(* IEC 61131-3 sources: F100R_S278_Temperville/MyController.device.xml.v3^/Plc Logic.plclogic.xml.v3^/Application.application.xml.v3^/06_Relógio, 3 files *)

(* ---- B_DataHora.prg.st ---- *)
PROGRAM B_DataHora
VAR
	LerDataHora: GetDateAndTime;
	SetDataHora: SetDateAndTime;
	TonAcertoHora: TON;
	TonAcertoHoraIn: BOOL;
	TonAcertoHoraQ: BOOL;
	uAnoRealTimeq_UIntMonth: UINT;
END_VAR

// Auto Acerto Data/Hora

TonAcertoHoraIn:= NOT TonAcertoHoraQ;

TonAcertoHora(IN:= TonAcertoHoraIn, PT:=T#30S , Q=>TonAcertoHoraQ, ET=> );

IF TonAcertoHoraQ THEN
	xAcertaRelogio:=TRUE;
END_IF

SetDataHora(
	i_xSetDateTime:= 	BtAcertaRelogioPlc,
	i_UIntYear:= 		uAcertoAno,
	i_UIntMonth:= 		uAcertoMes,
	i_UIntDay:= 		uAcertoDia,
	i_UIntHour:= 		uAcertoHora,
	i_UIntMinute:= 		uAcertoMinuto,
	i_UIntSecond:= 		uAcertoSegundo,
	q_UIntDatetoUTC_diag=> ,
	q_UIntRtcSet_diag=> );

IF BtAcertaRelogioPlc THEN
	BtAcertaRelogioPlc:=false;
END_IF

LerDataHora(
	q_UIntYear=> 		uAnoRealTime,
	q_UIntMonth=> 		uMesRealTime,
	q_UIntDay=> 		uDiaRealTime,
	q_UIntHour=> 		uHoraRealTime,
	q_UIntMinute=> 		uMinutoRealTime,
	q_UIntSecond=> 		uSegundoRealTime,
	q_UIntMSecond=> 	uMSegundoRealTime,
	q_UIntDayOfWeek=> 	uDiaSemanaRealTime,
	q_UIntYday=> 		uDiaAnoRealTime);

IF xRelogioAcertado THEN
	xAcertaRelogio:=FALSE;
	xRelogioAcertado:=FALSE;
END_IF

(* ---- C_ProgramacaoHoraria.prg.st ---- *)
PROGRAM C_ProgramacaoHoraria
VAR
	AtivaDesativaSemanal: HabilitaDesabilita;
	AtivaDesativaDiaria: HabilitaDesabilita;
	xLigaSegunda: BOOL;
	xLigaTerca: BOOL;
	xLigaQuarta: BOOL;
	xLigaQuinta: BOOL;
	xLigaSexta: BOOL;
	xLigaSabado: BOOL;
	xLigaDomingo: BOOL;
	xLigaSemanda: BOOL;

	xLigaHoraSeg: BOOL;
	xLigaMinutoSeg: BOOL;
	xLigaHoraTer: BOOL;
	xLigaMinutoTer: BOOL;
	xLigaHoraQua: BOOL;
	xLigaMinutoQua: BOOL;
	xLigaHoraQui: BOOL;
	xLigaMinutoQui: BOOL;
	xLigaHoraSex: BOOL;
	xLigaMinutoSex: BOOL;
	xLigaHoraSab: BOOL;
	xLigaMinutoSab: BOOL;
	xLigaHoraDom: BOOL;
	xLigaMinutoDom: BOOL;
	xLigaSegundo: BOOL;
	xLigaTempoSeg: BOOL;
	xLigaTempoTer: BOOL;
	xLigaTempoQua: BOOL;
	xLigaTempoQui: BOOL;
	xLigaTempoSex: BOOL;
	xLigaTempoSab: BOOL;
	xLigaTempoDom: BOOL;
	xLigaSemanaDias: BOOL;
	uDiaSemanaRealTimeAuxiliar: UINT;
	xAuxLiga: BOOL;
	xAuxEnable: BOOL;
	teste: BOOL;

	xDataHoraDomProgOk	: BOOL ;
	xDataHoraSegProgOk	: BOOL ;
	xDataHoraTerProgOk	: BOOL ;
	xDataHoraQuaProgOk	: BOOL ;
	xDataHoraQuiProgOk	: BOOL ;
	xDataHoraSexProgOk	: BOOL ;
	xDataHoraSabProgOk	: BOOL ;

END_VAR

// Programação Horario

IF uDiaSemanaRealTime=0 THEN
	uDiaSemanaRealTimeAuxiliar:=7;
ELSE
	uDiaSemanaRealTimeAuxiliar:=uDiaSemanaRealTime;
END_IF

//Horario Domingo
xLigaHoraDom:=		uHoraRealTime = rHorProgramadoDom;
xLigaMinutoDom:=	uMinutoRealTime = rMinProgramadoDom;
xLigaSegundo:=		uSegundoRealTime = uSegProgramado;
xLigaTempodom := xLigaHoraDom AND xLigaMinutoDom AND xLigaSegundo;

IF bDomingo AND uDiaSemanaRealTimeAuxiliar=7 THEN
	xLigaDomingo:=TRUE;
ELSE
	xLigaDomingo:=FALSE;
END_IF

xDataHoraDomProgOk:= xLigaDomingo AND xLigaTempodom;
IF xDataHoraDomProgOk THEN
	rTempoRampa03 := rRampaDomingo;
END_IF

//Horario Segunda
xLigaHoraSeg:=		uHoraRealTime = rHorProgramadoSeg;
xLigaMinutoSeg:=	uMinutoRealTime = rMinProgramadoSeg;
xLigaSegundo:=		uSegundoRealTime = uSegProgramado;
xLigaTempoSeg := xLigaHoraSeg AND xLigaMinutoSeg AND xLigaSegundo;

IF bSegunda AND uDiaSemanaRealTimeAuxiliar=1 THEN
	xLigaSegunda:=TRUE;
ELSE
	xLigaSegunda:=FALSE;
END_IF

xDataHoraSegProgOk:= xLigaSegunda AND xLigaTempoSeg;
IF xDataHoraSegProgOk THEN
	rTempoRampa03 := rRampaSegunda;
END_IF

//Horario Terça
xLigaHoraTer:=		uHoraRealTime = rHorProgramadoTer;
xLigaMinutoTer:=	uMinutoRealTime = rMinProgramadoTer;
xLigaSegundo:=		uSegundoRealTime = uSegProgramado;
xLigaTempoTer := xLigaHoraTer AND xLigaMinutoTer AND xLigaSegundo;

IF bTerca AND uDiaSemanaRealTimeAuxiliar=2 THEN
	xLigaTerca:=TRUE;
ELSE
	xLigaTerca:=FALSE;
END_IF

xDataHoraTerProgOk:= xLigaTerca AND xLigaTempoTer;
IF xDataHoraTerProgOk THEN
	rTempoRampa03 := rRampaTerca;
END_IF
//Horario Quarta
xLigaHoraQua:=		uHoraRealTime = rHorProgramadoQua;
xLigaMinutoQua:=	uMinutoRealTime = rMinProgramadoQua;
xLigaSegundo:=		uSegundoRealTime = uSegProgramado;
xLigaTempoQua := xLigaHoraQua AND xLigaMinutoQua AND xLigaSegundo;

IF bQuarta AND uDiaSemanaRealTimeAuxiliar=3 THEN
	xLigaQuarta:=TRUE;
ELSE
	xLigaQuarta:=FALSE;
END_IF

xDataHoraQuaProgOk:= xLigaQuarta AND xLigaTempoQua;
IF xDataHoraQuaProgOk THEN
	rTempoRampa03 := rRampaQuarta;
END_IF

//Horario Quinta
xLigaHoraQui:=		uHoraRealTime = rHorProgramadoQui;
xLigaMinutoQui:=	uMinutoRealTime = rMinProgramadoQui;
xLigaSegundo:=		uSegundoRealTime = uSegProgramado;
xLigaTempoQui := xLigaHoraQui AND xLigaMinutoQui AND xLigaSegundo;

IF bQuinta AND uDiaSemanaRealTimeAuxiliar=4 THEN
	xLigaQuinta:=TRUE;
ELSE
	xLigaQuinta:=FALSE;
END_IF

xDataHoraQuiProgOk:= xLigaQuinta AND xLigaTempoQui;
IF xDataHoraQuiProgOk THEN
	rTempoRampa03 := rRampaQuinta;
END_IF

//Horario Sexta
xLigaHoraSex:=		uHoraRealTime = rHorProgramadoSex;
xLigaMinutoSex:=	uMinutoRealTime = rMinProgramadoSex;
xLigaSegundo:=		uSegundoRealTime = uSegProgramado;
xLigaTempoSex := xLigaHoraSex AND xLigaMinutoSex AND xLigaSegundo;

IF bSexta AND uDiaSemanaRealTimeAuxiliar=5 THEN
	xLigaSexta:=TRUE;
ELSE
	xLigaSexta:=FALSE;
END_IF

xDataHoraSexProgOk:= xLigaSexta AND xLigaTempoSex;
IF xDataHoraSexProgOk THEN
	rTempoRampa03 := rRampaSexta;
END_IF

//Horario Sabado
xLigaHoraSab:=		uHoraRealTime = rHorProgramadoSab;
xLigaMinutoSab:=	uMinutoRealTime = rMinProgramadoSab;
xLigaSegundo:=		uSegundoRealTime = uSegProgramado;
xLigaTempoSab := 	xLigaHoraSab AND xLigaMinutoSab AND xLigaSegundo;

IF bSabado AND uDiaSemanaRealTimeAuxiliar=6 THEN
	xLigaSabado:=TRUE;
ELSE
	xLigaSabado:=FALSE;
END_IF

xDataHoraSabProgOk:= xLigaSabado AND xLigaTempoSab;
IF xDataHoraSabProgOk THEN
	rTempoRampa03 := rRampaSabado;
END_IF

// Programação Horaria Ativada

IF bDomingo OR bSegunda OR bTerca OR bQuarta OR bQuinta OR bSexta OR bSabado THEN
	bStatusAtvProgSemana:=TRUE;
ELSE
	bStatusAtvProgSemana:=FALSE;
END_IF

xStatusAtvProgHoraria:= bStatusAtvProgSemana;

// Liga Resisências

xDataHoraProgOk:= xDataHoraDomProgOk or xDataHoraSegProgOk OR xDataHoraTerProgOk OR xDataHoraQuaProgOk OR xDataHoraQuiProgOk OR xDataHoraSexProgOk OR xDataHoraSabProgOk;

(* ---- D_ProgramacaoTempo.prg.st ---- *)
PROGRAM D_ProgramacaoTempo
VAR
	xTrvAno: BOOL;
	xTrvMes: BOOL;
	xTrvDia: BOOL;
	xTrvData: BOOL;
	xTrvHora: BOOL;
	xTrvMinuto: BOOL;
	xTrvSegundo: BOOL;
	xTrvTempo: BOOL;
	xTrava: BOOL;
END_VAR

IF BtHabDesabBloqueio THEN
	IF xBloqueioHabilitado THEN
		xBloqueioHabilitado:=FALSE;
	ELSE
		xBloqueioHabilitado:=TRUE;
	END_IF
	BtHabDesabBloqueio:=FALSE;
END_IF

xTrvAno:=	uAnoRealTime = uAnoProgTrv;// = 2015;
xTrvMes:=	uMesRealTime = uMesProgTrv;// = 5;
xTrvDia:=	uDiaRealTime = uDiaProgTrv;// = 10;
xTrvData := xTrvAno AND xTrvMes AND xTrvDia;

xTrvHora:=		uHoraRealTime = uHorProgTrv;// = 23;
xTrvMinuto:=	uMinutoRealTime = uMinProgTrv;// = 0;
xTrvSegundo:=	uSegundoRealTime = uSegProgTrv;// = 0;
xTrvTempo := xTrvHora AND xTrvMinuto AND xTrvSegundo ;

xTrava:= xTrvData AND xTrvTempo AND xBloqueioHabilitado;

IF xTrava THEN
	xSeguranca:=TRUE;
END_IF
IF BtDesbloqueio THEN
	xSeguranca:=FALSE;
	BtDesbloqueio:=FALSE;
END_IF
